// TIA Portal V16 program export: 0 tag tables, 1 data types, 2 data blocks, 5 code blocks (in call order from the OBs), 1 instance data blocks

TYPE "Point"
// stored: CreationDate 2020-12-17T10:41:14.5497731Z, InterfaceModifiedDate 2020-12-17T10:41:40.9176599Z, IsConsistent true, IsFailsafeCompliant false, IsKnowHowProtected false, LibraryConformanceStatus The object is library-conformant., ModifiedDate 2020-12-17T10:41:54.4302381Z
   STRUCT
      x { S7_SetPoint := 'True'} : Int := 100;
      y { S7_SetPoint := 'True'} : Int := 100;
   END_STRUCT;
END_TYPE

DATA_BLOCK "Data_block_1"   // DB1
{ S7_Optimized_Access := 'TRUE' }
VERSION : 0.1
// stored: AutoNumber true, DBAccessibleFromOPCUA true, IsOnlyStoredInLoadMemory false, IsRetainMemResEnabled false, IsWriteProtectedInAS false, MemoryReserve 100
   VAR
      VarI1 : Int;
      VarI2 { ExternalVisible := 'False'} : Int;
      VarI3 { ExternalVisible := 'False'; ExternalWritable := 'False'} : Int;
      VarI4 { ExternalAccessible := 'False'; ExternalVisible := 'False'; ExternalWritable := 'False'} : Int;
   END_VAR
BEGIN
END_DATA_BLOCK

DATA_BLOCK "Data_block_2"   // DB3
{ S7_Optimized_Access := 'TRUE' }
VERSION : 0.1
// stored: AutoNumber true, CodeModifiedDate 2020-12-17T10:42:33.3081896Z, CompileDate 2020-12-17T10:42:38.4660302Z, CreationDate 2020-12-17T10:42:13.2923269Z, DBAccessibleFromOPCUA true, DownloadWithoutReinit false, InterfaceModifiedDate 2020-12-17T10:42:33.3081896Z, IsConsistent true, IsKnowHowProtected false, IsOnlyStoredInLoadMemory false, IsPLCDB false, IsRetainMemResEnabled false, IsWriteProtectedInAS false, MemoryReserve 100, ModifiedDate 2020-12-17T10:42:33.3081896Z, ParameterModified 2020-12-17T10:42:33.3081896Z, StructureModified 2020-12-17T10:42:33.3081896Z
   VAR
      p1 { S7_SetPoint := 'True'} : "Point";
   END_VAR
   VAR RETAIN
      p2 { S7_SetPoint := 'True'} : "Point";
   END_VAR
   VAR
      p3 { S7_SetPoint := 'True'} : "Point";
   END_VAR
   VAR RETAIN
      p4 { S7_SetPoint := 'True'} : "Point";
   END_VAR
BEGIN
END_DATA_BLOCK

ORGANIZATION_BLOCK "Main"   // OB1, LAD, ProgramCycle
TITLE = "Main Program Sweep (Cycle)"
{ S7_Optimized_Access := 'TRUE' }
VERSION : 0.1
// stored: AutoNumber true, IsIECCheckEnabled false, SetENOAutomatically false
   VAR_INPUT
      Initial_Call : Bool;   // Initial call of this OB
      Remanence : Bool;   // =True, if remanent data are available
   END_VAR
BEGIN

REGION Network 1
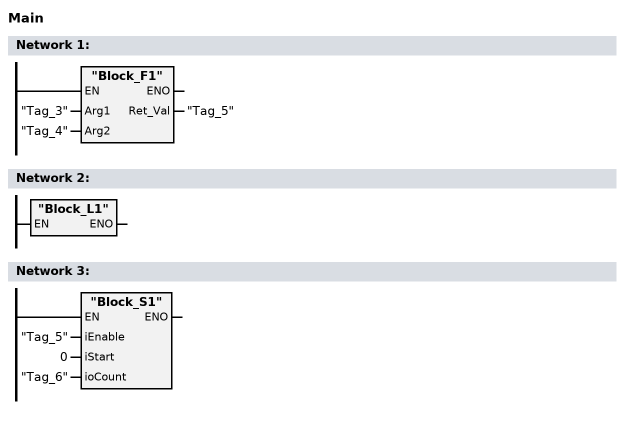
   RUNG wire#powerrail
      "Block_F1"(Arg1 := "Tag_3", Arg2 := "Tag_4", Ret_Val => "Tag_5")
   END_RUNG
   // the same network as SCL:
   "Tag_5" := "Block_F1"(Arg1 := "Tag_3", Arg2 := "Tag_4");
END_REGION

REGION Network 2
   RUNG wire#powerrail
      "Block_L1"()
   END_RUNG
   // the same network as SCL:
   "Block_L1"();
END_REGION

REGION Network 3
   RUNG wire#powerrail
      "Block_S1"(iEnable := "Tag_5", iStart := 0, ioCount := "Tag_6")
   END_RUNG
   // the same network as SCL:
   "Block_S1"(iEnable := "Tag_5", iStart := 0, ioCount := "Tag_6");
END_REGION
END_ORGANIZATION_BLOCK

FUNCTION "Block_F1" : Bool   // FC2, FBD
TITLE = XOR function
{ S7_Optimized_Access := 'TRUE' }
VERSION : 0.1
// As an example
// stored: AutoNumber true, IsIECCheckEnabled false, SetENOAutomatically false, UDAEnableTagReadback false
   VAR_INPUT
      Arg1 : Bool;
      Arg2 : Bool;
   END_VAR
BEGIN

REGION Network 1: N1
   // Body
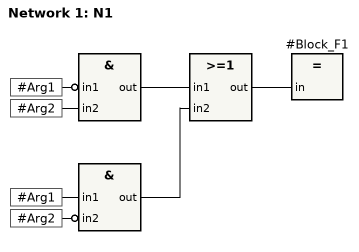
   #Block_F1 := (NOT #Arg1 AND #Arg2) OR (#Arg1 AND NOT #Arg2);
END_REGION
END_FUNCTION

FUNCTION "Block_L1" : Void   // FC1, LAD
{ S7_Optimized_Access := 'TRUE' }
VERSION : 0.1
// stored: AutoNumber true, IsIECCheckEnabled false, SetENOAutomatically false, UDAEnableTagReadback false
   VAR_TEMP
      Tag_1 : Bool;
      Tag_2 : Bool;
   END_VAR
BEGIN

REGION Network 1
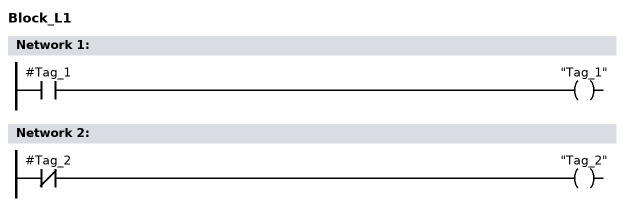
   RUNG wire#powerrail
      Contact( #Tag_1 )
      Coil( "Tag_1" )
   END_RUNG
   // the same network as SCL:
   "Tag_1" := #Tag_1;
END_REGION

REGION Network 2
   RUNG wire#powerrail
      I_Contact( #Tag_2 )
      Coil( "Tag_2" )
   END_RUNG
   // the same network as SCL:
   "Tag_2" := NOT #Tag_2;
END_REGION
END_FUNCTION

FUNCTION "Block_S1" : Void   // FC3, SCL
{ S7_Optimized_Access := 'TRUE' }
// stored: CodeModifiedDate 2020-12-17T10:18:16.964766Z, CompileDate 2020-12-17T10:18:16.964766Z, CreationDate 2020-12-17T10:17:02.6275941Z, InterfaceModifiedDate 2020-12-17T10:17:32.4776481Z, IsConsistent true, LibraryConformanceStatus The object is library-conformant., ModifiedDate 2020-12-17T10:18:16.964766Z, ParameterModified 2020-12-17T10:17:32.4776481Z, SetENOAutomatically false, StructureModified 2020-12-17T10:17:32.4776481Z
   VAR_INPUT
      iEnable : Bool;
      iStart : Int;
   END_VAR
   VAR_IN_OUT
      ioCount : Int;
   END_VAR
BEGIN
   IF #iEnable THEN
       #ioCount := #ioCount + 1;
   ELSE
       #ioCount := #iStart;
   END_IF;
END_FUNCTION

FUNCTION_BLOCK "XBlock_1"   // FB1, FBD
{ S7_Optimized_Access := 'TRUE' }
VERSION : 0.1
// stored: AutoNumber true, IsIECCheckEnabled false, IsRetainMemResEnabled false, MemoryReserve 100, SetENOAutomatically false, UDAEnableTagReadback false
   VAR_INPUT
      iEnable : Bool;
      iStart : Int;
   END_VAR
   VAR_OUTPUT
      qCounter : Int;
   END_VAR
   VAR
      sCounter : Int;
   END_VAR
   VAR CONSTANT
      C_ADD : Int := 1;
   END_VAR
BEGIN

REGION Network 1
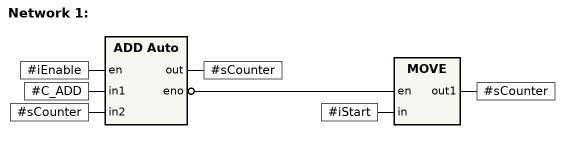
   IF #iEnable THEN #sCounter := #C_ADD + #sCounter; END_IF;
   IF NOT #iEnable THEN #sCounter := #iStart; END_IF;
END_REGION
END_FUNCTION_BLOCK

DATA_BLOCK "XBlock_1_DB"   // DB2
{ S7_Optimized_Access := 'TRUE' }
VERSION : 0.1
// stored: AutoNumber true, CodeModifiedDate 2020-12-17T10:30:13.4748899Z, CompileDate 2020-12-17T10:32:57.5038962Z, CreationDate 2020-12-17T10:30:13.3967342Z, DBAccessibleFromOPCUA true, DownloadWithoutReinit false, InstanceOfName XBlock_1, InstanceOfNumber 1, InstanceOfType FB, InterfaceModifiedDate 2020-12-17T10:28:41.3528478Z, IsConsistent true, IsKnowHowProtected false, IsRetainMemResEnabled false, MemoryReserve 100, ModifiedDate 2020-12-17T10:30:13.4748899Z, ParameterModified 2020-12-17T10:28:41.3528478Z, StructureModified 2020-12-17T10:28:41.3528478Z, UDAEnableTagReadback false
"XBlock_1"
BEGIN
END_DATA_BLOCK
